// TIA Portal V19 export
DATA_BLOCK "SCALE_SET"   // DB36
{ S7_Optimized_Access := 'FALSE' }
   VAR RETAIN
      CT_SCALE_MIN : Real;
      CT_SCALE_MAX : Real;
      PH_SCALE_MIN : Real;
      PH_SCALE_MAX : Real;
      TS_SCALE_MIN : Real;
      TS_SCALE_MAX : Real;
      CT_NORM : Real;
      PH_NORM : Real;
      TS_NORM : Real;
      CT_PV : Real;
      PH_PV : Real;
      TS_PV : Real;
      FWD_PUMP_SPEED : Real;
      HYSTERSIS : Real;
      "PUMP-1_MIN_SPEED" : Int;
      "PUMP-1_MAX_SPEED" : Int;
   END_VAR
BEGIN
END_DATA_BLOCK
